{attribute 'linkalways'} 
{attribute 'no_explicit_call' := 'This FB is a CLASS and must be accessed using methods or properties'}
{attribute 'enable_dynamic_creation'}
FUNCTION_BLOCK Node_F_VN_BitwiseXorVectorWithImage EXTENDS VisionNode
VAR
    aVector : _TcVnVector4_LREAL;
    ipSrcImage : _ITcVnImage;
    ipDestImage : _ITcVnImage;
    hrPrev : _HRESULT(S_OK);
	hresult : _HRESULT(S_OK);
END_VAR

METHOD PUBLIC  Clone : I_Node
VAR
	pNode : POINTER TO Node_F_VN_BitwiseXorVectorWithImage;
END_VAR
pNode := __NEW(Node_F_VN_BitwiseXorVectorWithImage);
Clone := pNode^;
END_METHOD

METHOD FB_init : BOOL
VAR_INPUT
	bInitRetains : BOOL; // if TRUE, the retain variables are initialized (warm start / cold start)
	bInCopyCode : BOOL;  // if TRUE, the instance afterwards gets moved into the copy code (online change)
END_VAR
AddInput('aVector', aVector);
AddInput('ipSrcImage', ipSrcImage);
AddInput('hrPrev', hrPrev);
AddOutput('ipDestImage', ipDestImage);
AddOutput('hresult',hresult);
END_METHOD

METHOD PROTECTED OnExecute
hresult.Value := F_VN_BitwiseXorVectorWithImage(
    aVector := aVector.Value,
    ipSrcImage := ipSrcImage.Value,
	ipDestImage := ipDestImage.Value,
	hrPrev:= hrPrev.Value);
END_METHOD

METHOD PUBLIC PreExecutionCheck
VAR_INPUT
	Check : I_PreExecutionChecks;
END_VAR
Check.IsTrue(ipSrcImage.IsValid, 'ipSrcImage must contain an image');
END_METHOD

END_FUNCTION_BLOCK

(* stored: Version 1.1.0.1, ProductVersion 3.1.4024.13
   POU Node_F_VN_BitwiseXorVectorWithImage: Id {54a6b4fc-a2c8-02c9-090c-460f2aca326e}, SpecialFunc None
   Folder Constructor: Id {fbb72692-821a-0fc7-3787-29e0cd2219b1}
   Method Clone: Id {196a613c-fa4a-00ed-2963-f43555e5b243}
   Method FB_init: Id {c581e096-606b-0c9d-2050-0924d8acbc7e}
   Method OnExecute: Id {00b1366e-ed71-0c7f-1766-67823f1d1bdc}
   Method PreExecutionCheck: Id {72d20791-0803-048c-1aca-fc7c6421dd15} *)
